FUNCTION_BLOCK FB_Fenster
VAR_INPUT
	Freigabe_auto			: BOOL;
	Freigabe_Deakt_auto		: BOOL;
	Fenster_AUF				: BOOL;
	Fenster_ZU				: BOOL;
	Quittierung				: BOOL;
	Parameter_init			: ST_Fenster_Parameter;

END_VAR
VAR_OUTPUT
	{attribute 'OPC.UA.DA' := '1'}Parameter				: ST_Fenster_Parameter;		
	{attribute 'OPC.UA.DA' := '1'}Steuerung				: ST_Fenster_Steuerung;		
	{attribute 'OPC.UA.DA' := '1'}Stellwert				: ST_Fenster_Stellwert;		
	{attribute 'OPC.UA.DA' := '1'}Zustand					: ST_Fenster_Zustand;	
END_VAR
VAR

	OUT_SERVO_Fenster_Halle_AUF					AT %Q*: BOOL;
	OUT_SERVO_Fenster_Halle_ZU					AT %Q*: BOOL;

	LeseDaten			: FB_Fenster_Input;
	QuitTrig			: FB_SetResetFallTrigger;
	Zustandscheck		: FB_Fenster_Zustandscheck;
	Logik				: FB_Fenster_Logik;
	SchreibeDaten		: FB_Fenster_Output;


	Ablaufsteuerung: FB_Fenster_Ablaufsteuerung;
END_VAR

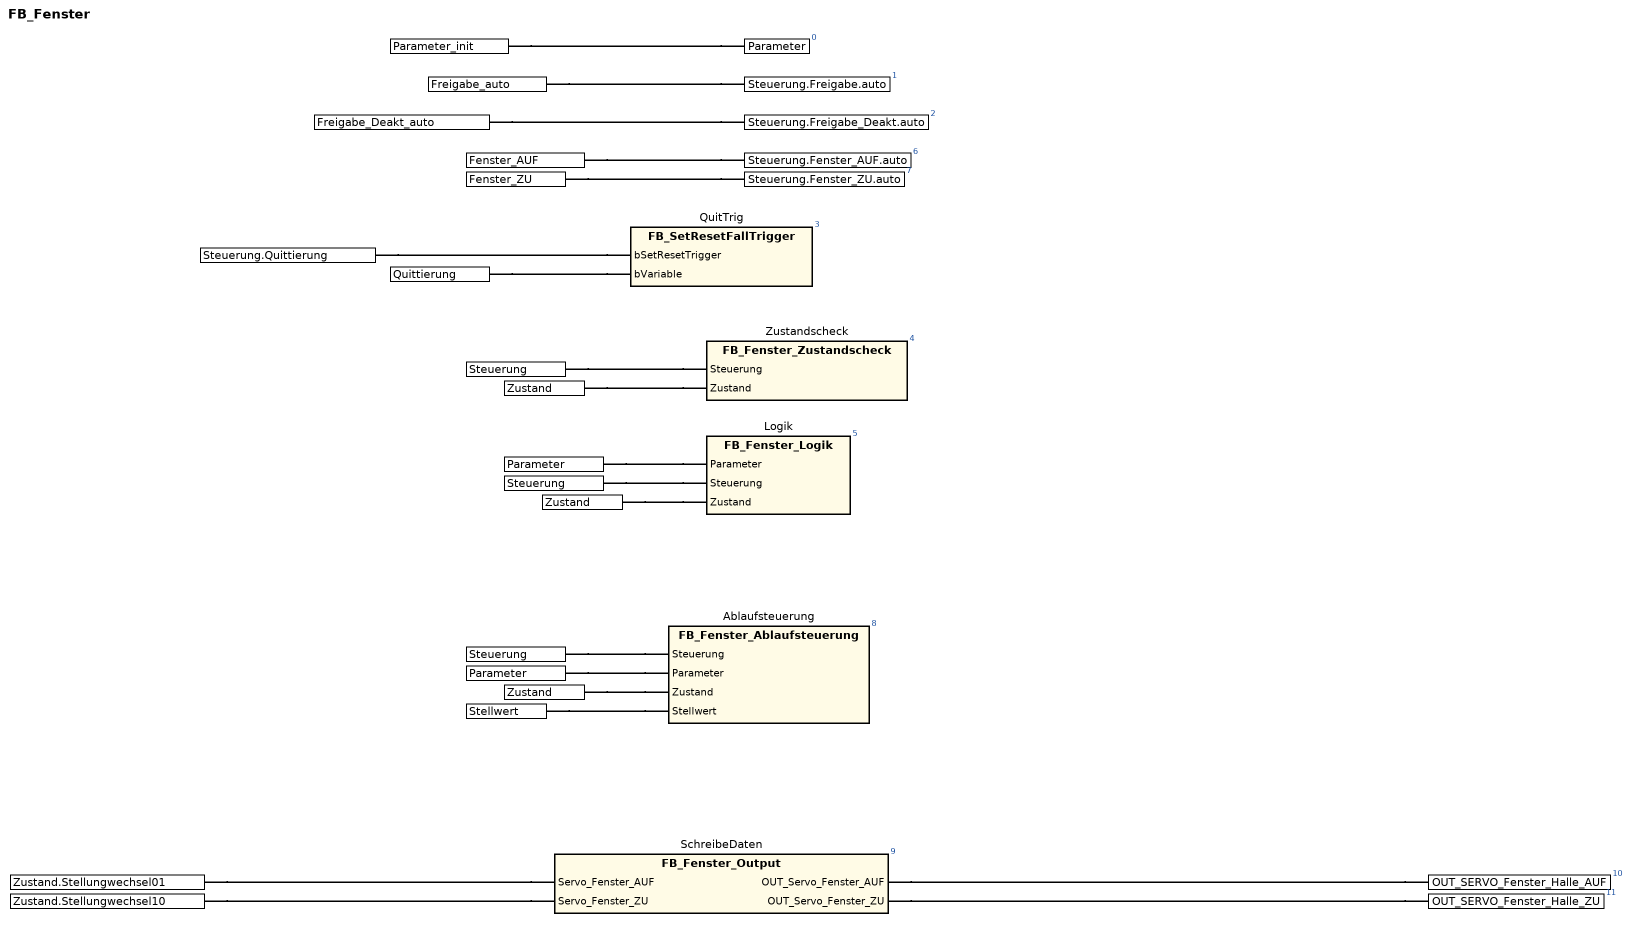
Parameter := Parameter_init;
Steuerung.Freigabe.auto := Freigabe_auto;
Steuerung.Freigabe_Deakt.auto := Freigabe_Deakt_auto;
QuitTrig(bSetResetTrigger := Steuerung.Quittierung, bVariable := Quittierung); // FB_SetResetFallTrigger
Zustandscheck(Steuerung := Steuerung, Zustand := Zustand); // FB_Fenster_Zustandscheck
Logik(Parameter := Parameter, Steuerung := Steuerung, Zustand := Zustand); // FB_Fenster_Logik
Steuerung.Fenster_AUF.auto := Fenster_AUF;
Steuerung.Fenster_ZU.auto := Fenster_ZU;
Ablaufsteuerung(Steuerung := Steuerung, Parameter := Parameter, Zustand := Zustand, Stellwert := Stellwert); // FB_Fenster_Ablaufsteuerung
SchreibeDaten(Servo_Fenster_AUF := Zustand.Stellungwechsel01, Servo_Fenster_ZU := Zustand.Stellungwechsel10); // FB_Fenster_Output
OUT_SERVO_Fenster_Halle_AUF := SchreibeDaten.OUT_Servo_Fenster_AUF;
OUT_SERVO_Fenster_Halle_ZU := SchreibeDaten.OUT_Servo_Fenster_ZU;

END_FUNCTION_BLOCK

(* stored: Version 1.1.0.1, ProductVersion 3.1.4024.9
   POU FB_Fenster: Id {8aa21112-dc64-4a6c-8e23-be54f2c3c386}, SpecialFunc None *)
